PROGRAM PRG_LVCP2_Group3
VAR
    // Function Block Instance
    fbContactor: FB_ContactorControl;

    // Contactor 1 IO Structure  
    stContactor_IO: ST_ContactorIO;
    
    // Başlangıç konfigürasyonu için flag
    bContactorInitDone: BOOL := FALSE;
    bCapacitorInitDone: BOOL := FALSE;	
END_VAR



	M_Contactor();
	
	M_Capacitor();

METHOD M_Capacitor : BOOL
VAR
    nGroupIndex : INT;
END_VAR

nGroupIndex := 2;  // Grup 3 için index

IF NOT bCapacitorInitDone THEN
    // Grup 3 değerlerini ata
    GVL_LVCP2.astCompensationGroups[nGroupIndex].rPower := 25.0;
    GVL_LVCP2.astCompensationGroups[nGroupIndex].rVoltage := 450.0;
    GVL_LVCP2.astCompensationGroups[nGroupIndex].nQuantity := 6;
    GVL_LVCP2.astCompensationGroups[nGroupIndex].sTagPrefix := '+EP7-22C1';
    GVL_LVCP2.astCompensationGroups[nGroupIndex].sProductCode := 'ENT.CXD-450-25';
    
    bCapacitorInitDone := TRUE;
END_IF

// Grup 3 aktif durumu
GVL_LVCP2.abGroupActive[nGroupIndex] := stContactor_IO.bFeedback;

M_Capacitor := TRUE;
END_METHOD

METHOD M_Contactor : BOOL
VAR_INPUT
END_VAR
IF NOT bContactorInitDone THEN
    // Konfigürasyon parametreleri
    GVL_LVCP2.stGroup3_ContactorHMI.stConfig.sProjectCode := '+EP7-23K1';
    GVL_LVCP2.stGroup3_ContactorHMI.stConfig.sProductCode := 'ABB-1SFL597001R7011';
    GVL_LVCP2.stGroup3_ContactorHMI.stConfig.rRatedCurrent := 500.0;
    GVL_LVCP2.stGroup3_ContactorHMI.stConfig.rRatedVoltage := 1000.0;
    GVL_LVCP2.stGroup3_ContactorHMI.stConfig.nPhaseCount := 3;
    GVL_LVCP2.stGroup3_ContactorHMI.stConfig.tFeedbackDelay := T#500MS;
    GVL_LVCP2.stGroup3_ContactorHMI.stConfig.tWeldedDelay := T#2S;
    GVL_LVCP2.stGroup3_ContactorHMI.stConfig.dwOperationLimit := 100000;
    
    // Başlangıç bakım sayacı
    GVL_LVCP2.stGroup3_ContactorHMI.stStatistics.dwRemainingOperations := GVL_LVCP2.stGroup3_ContactorHMI.stConfig.dwOperationLimit;
    
    bContactorInitDone := TRUE;
END_IF

// Function Block Çağrısı
fbContactor(
    // Fiziksel Girişler
    bFeedback := stContactor_IO.bFeedback,
    bPLCControl := stContactor_IO.bPLCControl,
    
    // Güvenlik Girişleri
    bSafetyLoop := GVL_Alarm.bSafetyLoop,
    bInterlock := FALSE,
    
    // Sistem Girişleri
    bMasterReset := GVL_Alarm.bMasterReset,
    
    // HMI Bağlantısı
    stHMI := GVL_LVCP2.stGroup3_ContactorHMI,
    
    // Fiziksel Çıkış
    bOutput => stContactor_IO.bOutput
);

M_Contactor := TRUE;
END_METHOD

END_PROGRAM

(* stored: Version 1.1.0.1, ProductVersion 3.1.4024.14
   POU PRG_LVCP2_Group3: Id {bb8d8cc4-ba78-49cb-89e8-b50f4c03cc33}, SpecialFunc None
   Method M_Capacitor: Id {13e12990-f9e8-4cd9-b4ee-b5dc0c0172ce}
   Method M_Contactor: Id {9d83fe14-1321-4b28-ab23-2e06add99fb1} *)
